INTERFACE ITF_Regelschuif_OutClose_DG

METHOD set : BOOL
VAR_INPUT
	state : BOOL;	
END_VAR
END_METHOD

END_INTERFACE

(* stored: Version 1.1.0.1, ProductVersion 3.1.4026.8
   Itf ITF_Regelschuif_OutClose_DG: Id {698377fc-52e7-4146-bb11-263afae30f9b}
   Method set: Id {ed471539-1287-41e7-aa70-cccf91c5f86d} *)
